PROGRAM p09_timers
VAR
	pulseTimer: TP;
	onDelayTimer: TON;
	offDelayTimer: TOF;
	ptValue: TIME;
	ontValue: TIME;
	oftValue: TIME;
	S0: BOOL;	
	L0: BOOL;
	L1: BOOL;
	L2: BOOL;
END_VAR

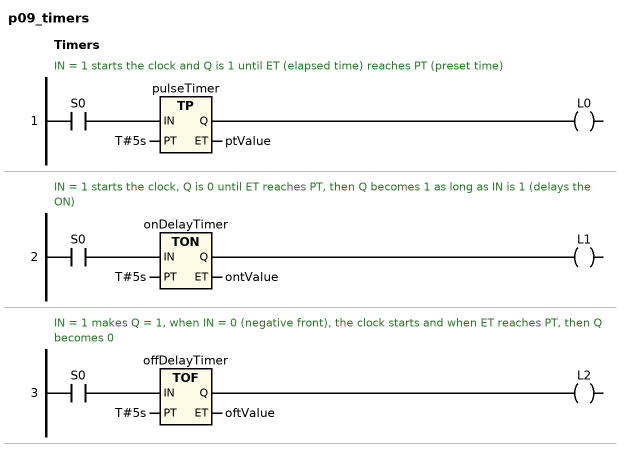
// NETWORK 1: Timers
// IN = 1 starts the clock and Q is 1 until ET (elapsed time) reaches PT (preset time)
pulseTimer(IN := S0, PT := T#5s, ET => ptValue); // TP
L0 := pulseTimer.Q;

// NETWORK 2
// IN = 1 starts the clock, Q is 0 until ET reaches PT, then Q becomes 1 as long as IN is 1 (delays the ON)
onDelayTimer(IN := S0, PT := T#5s, ET => ontValue); // TON
L1 := onDelayTimer.Q;

// NETWORK 3
// IN = 1 makes Q = 1, when IN = 0 (negative front), the clock starts and when ET reaches PT, then Q becomes 0
offDelayTimer(IN := S0, PT := T#5s, ET => oftValue); // TOF
L2 := offDelayTimer.Q;

END_PROGRAM

(* stored: Version 1.1.0.1, ProductVersion 3.1.4024.13
   POU p09_timers: Id {ee744d0c-41fe-4cb3-992c-2546a4341f8c}, SpecialFunc None *)
